# EPICS substitutions: db/Beckhoff_7XXX/ecmcEP7041-0000.substitutions
file "ecmcEL5042-chX.template"
{
  pattern {CH_ID}
          {01   }
}
